PROGRAM MAIN
VAR
	So_Taktgenerator				: FB_Zentral_TaktimpulsGenerator; 
	
	Sx_Takt			: BOOL; 
	Sx_Impuls		: BOOL; 
	Si_Counter		: INT; 
	
END_VAR


So_Taktgenerator(Ir_Frequenz := 1.0, Ox_Takt => Sx_Takt, Ox_Impuls => Sx_Impuls); 

IF(Sx_Impuls) THEN 
	Si_Counter := Si_Counter + 1;
END_IF

END_PROGRAM

(* stored: Version 1.1.0.1, ProductVersion 3.1.4024.9
   POU MAIN: Id {bdaa0c53-7414-42f8-b710-e526f3e6d41b}, SpecialFunc None *)
